FUNCTION INTERNAL Power : LREAL
VAR_INPUT
  v : LREAL;
  e : LREAL;
END_VAR

Power := SEL(v < 0, 1.0, -1.0) * EXPT(ABS(v), e);

END_FUNCTION

(* stored: Version 1.1.0.1, ProductVersion 3.1.4024.9
   POU Power: Id {76716193-d546-414d-a8ab-5cbcfa9a3d68}, SpecialFunc None *)
